INTERFACE ITF_MQTTTool

METHOD SendMQTTMessage : BOOL
VAR_INPUT
	Status : STRING;
END_VAR
END_METHOD

END_INTERFACE

(* stored: Version 1.1.0.1, ProductVersion 3.1.4024.12
   Itf ITF_MQTTTool: Id {fd375ca1-9267-486b-b188-2cebefbc230b}
   Method SendMQTTMessage: Id {d3655495-1523-4000-8737-af976150ac0b} *)
